TYPE ST_LOG_Alarms :
STRUCT

	nAlarmCounter				: UINT;
	sTotalAlarmTime				: T_TimeLog;
	sMaxAlarmTime				: T_TimeLog;
	stMaxAlarmTimeStamp			: TIMESTRUCT;

END_STRUCT
END_TYPE

(* stored: Version 1.1.0.1
   DUT ST_LOG_Alarms: Id {c6ee3c42-7caa-4d94-ae62-d8f452e07943} *)
